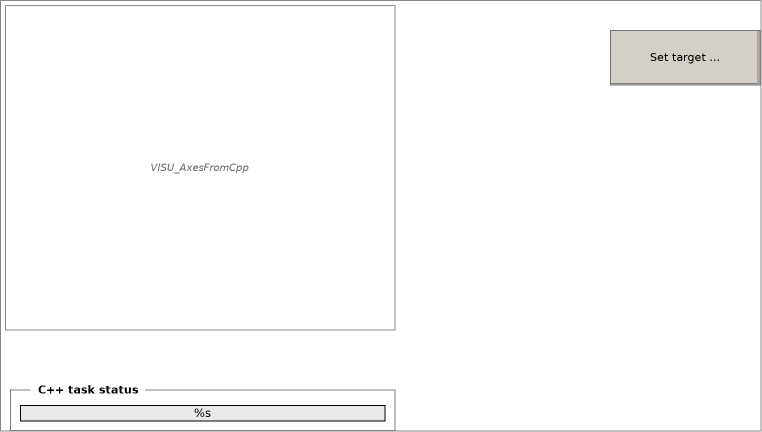
VISUALIZATION VISU_AxesTarget  // 762x432
VAR_IN_OUT
	ref : Axes;
    widget : AxesWidget;
END_VAR
    Polyline (30,390) (10,390) (10,430) (395,430) (395,390) (145,390)
    Rectangle (20,405 365x16), "%s", text variable: widget.cppAxesErrorString
    Label (35,380 115x20), "C++ task status"
    Frame (5,5 390x325)
        shows VISU_AxesFromCpp(ref := ref, widget := widget)
    Button (610,30 150x55), "Set target ..."
        OnMouseClick: OpenDialog Dialog=VISU_AxesSetTargetDialog, OpenModal=True, OpenCentered=True
END_VISUALIZATION

(* stored: Version 1.1.0.1, ProductVersion 3.1.4019.2
   Visu VISU_AxesTarget: Id {c6baf819-4cb1-43b7-ba9e-404e0a726958} *)
